// TIA Portal V17 export
// export: Created 2023-02-14T02:49:53.8743835Z, ExportSetting WithDefaults, DisplayName Totally Integrated Automation Portal, DisplayVersion V17, DisplayName TIA Portal Openness, DisplayVersion V17, DisplayName TIA Portal Teamcenter Gateway, DisplayVersion V17, DisplayName TIA Portal Version Control Interface, DisplayVersion V17, DisplayName SINAMICS Startdrive Advanced, DisplayVersion V17, DisplayName SINAMICS Startdrive G130, G150, S120, S150, SINAMICS MV, S210, DisplayVersion V17, DisplayName SINAMICS Startdrive G110M, G120, G120C, G120D, G120P, G115D, DisplayVersion V17, DisplayName STEP 7 Professional, DisplayVersion V17, DisplayName STEP 7 Safety, DisplayVersion V17, DisplayName WinCC Professional, DisplayVersion V17
VAR_GLOBAL   // PLC tag table "RIO Homomixer Panel"
   "FT-12.01 Pulse" AT %I6.0 : Bool;   // PULSE FLOW METER PROCESS WATER
   "FT-12.02 Pulse" AT %I6.1 : Bool;   // PULSE FLOW METER HOT WATER
   "FT-12.01 Flowrate" AT %IW7 : Int;   // FLOW METER PROCESS WATER
   "FT-12.02 Flowrate" AT %IW9 : Int;   // FLOW METER HOT WATER
   "Homo spare 18" AT %IW11 : Int;
   "Homo spare 19" AT %IW13 : Int;
   "ZSC-12.01" AT %I4.0 : Bool;   // INLET PROCESS WATER HOMOMIXER T-12.00 VALVE CLOSE POSITION
   "ZSC-12.02" AT %I4.1 : Bool;   // INLET HOT WATER HOMOMIXER T-12.00 VALVE CLOSE POSITION
   "ZSC-13.01" AT %I4.2 : Bool;   // INLET PROCESS WATER HOMOMIXER T-13.00 VALVE CLOSE POSITION
   "ZSC-13.02" AT %I4.3 : Bool;   // INLET HOT WATER HOMOMIXER T-13.00 VALVE CLOSE POSITION
   "LL-12.01" AT %I4.4 : Bool;   // LOW LEVEL SENSOR HOMOMIXER T-12.00
   "LL-13.01" AT %I4.5 : Bool;   // LOW LEVEL SENSOR HOMOMIXER T-13.00
   "ES1 Homomixer" AT %I4.6 : Bool;   // EMERGENCY STOP RIO HOMOMIXER
   "PS-01 Homomixer" AT %I4.7 : Bool;   // PRESURE SWITCH PNEUMATIC VALVE
   "ZSC-14.01" AT %I5.0 : Bool;   // MAIN CIP SUPPLY HOMOMIXER T-14.00 VALVE CLOSE POSITION
   "ZSC-14.02" AT %I5.1 : Bool;   // MAIN CIP SUPPLY LINE HOMOMIXER T-14.00 VALVE CLOSE POSITION
   "LL-14.01" AT %I5.2 : Bool;   // LOW LEVEL SENSOR HOMOMIXER T-14.00
   "Homo spare 01" AT %I5.3 : Bool;
   "Homo spare 02" AT %I5.4 : Bool;
   "Homo spare 03" AT %I5.5 : Bool;
   "Homo spare 04" AT %I5.6 : Bool;
   "Homo spare 05" AT %I5.7 : Bool;
   "Homo spare 06" AT %I6.2 : Bool;
   "Homo spare 07" AT %I6.3 : Bool;
   "Homo spare 08" AT %I6.4 : Bool;
   "Homo spare 09" AT %I6.5 : Bool;
   "Homo spare 10" AT %I6.6 : Bool;
   "Homo spare 11" AT %I6.7 : Bool;
   "Start/Stop P-12.01" AT %Q2.0 : Bool;   // START/STOP DIAPHRAGM PUMP HOMOMIXER T-12.00
   "Start/Stop P-13.01" AT %Q2.1 : Bool;   // START/STOP DIAPHRAGM PUMP HOMOMIXER T-13.00
   "Start/Stop P-14.01" AT %Q2.2 : Bool;   // START/STOP DIAPHRAGM PUMP HOMOMIXER T-14.00
   "Homo spare 13" AT %Q2.3 : Bool;
   "Homo spare 14" AT %Q2.4 : Bool;
   "Homo spare 15" AT %Q2.5 : Bool;
   "Homo spare 16" AT %Q2.6 : Bool;
   "Homo spare 17" AT %Q2.7 : Bool;
   "AV-12.01" AT %Q22.0 : Bool;   // AUTO BUTTERFLY VALVE PW INLET TO HOMOMIXER T-12.00
   "AV-12.02" AT %Q22.1 : Bool;   // AUTO BUTTERFLY VALVE HOT WATER INLET TO HOMOMIXER T-12.00
   "AV-12.03" AT %Q22.2 : Bool;   // AUTO BUTTERFLY VALVE OUTLET FROM HOMOMIXER T-12.00
   "AV-12.04" AT %Q22.3 : Bool;   // AUTO BUTTERFLY VALVE CIP SUPPLY LINE T-12.00 FROM DP-12.01
   "AV-12.05" AT %Q22.4 : Bool;   // AUTO BUTTERFLY VALVE CIP RETURN FROM HOMOMIXER T-12.00
   "AV-12.06" AT %Q22.5 : Bool;   // AUTO BUTTERFLY VALVE BYPASS DIAPRAGM PUMP P-12.01
   "AV-12.07" AT %Q22.6 : Bool;   // AUTO BUTTERFLY VALVE CIP SUPPLY HOMOMIXER T-12.00
   "AV-12.11" AT %Q22.7 : Bool;   // AUTO BUTTERFLY VALVE MAIN CIP SUPPLY LINE 1 HOMOMIXER T-12.00
   "AV-12.12" AT %Q23.0 : Bool;   // AUTO BUTTERFLY VALVE MAIN CIP SUPPLY LINE 1 HOT WATER T-01.00
   "AV-13.01" AT %Q23.1 : Bool;   // AUTO BUTTERFLY VALVE PW INLET TO HOMOMIXER T-13.00
   "AV-13.02" AT %Q23.2 : Bool;   // AUTO BUTTERFLY VALVE HOT WATER INLET TO HOMOMIXER T-13.00
   "AV-13.03" AT %Q23.3 : Bool;   // AUTO BUTTERFLY VALVE OUTLET FROM HOMOMIXER T-13.00
   "AV-13.04" AT %Q23.4 : Bool;   // AUTO BUTTERFLY VALVE CIP SUPPLY LINE T-13.00 FROM DP-12.01
   "AV-13.05" AT %Q23.5 : Bool;   // AUTO BUTTERFLY VALVE CIP RETURN FROM HOMOMIXER T-13.00
   "AV-13.06" AT %Q23.6 : Bool;   // AUTO BUTTERFLY VALVE BYPASS DIAPRAGM PUMP P-13.01
   "AV-13.07" AT %Q23.7 : Bool;   // AUTO BUTTERFLY VALVE CIP SUPPLY HOMOMIXER T-13.00
   "AV-14.01" AT %Q24.0 : Bool;   // AUTO BUTTERFLY VALVE PW INLET TO HOMOMIXER T-14.00
   "AV-14.02" AT %Q24.1 : Bool;   // AUTO BUTTERFLY VALVE HOT WATER INLET TO HOMOMIXER T-14.00
   "AV-14.03" AT %Q24.2 : Bool;   // AUTO BUTTERFLY VALVE OUTLET FROM HOMOMIXER T-14.00
   "AV-14.04" AT %Q24.3 : Bool;   // AUTO BUTTERFLY VALVE CIP SUPPLY LINE T-14.00 CIP SUPPLY LINE 1
   "AV-14.05" AT %Q24.4 : Bool;   // AUTO BUTTERFLY VALVE CIP RETURN FROM HOMOMIXER T-14.00
   "AV-14.06" AT %Q24.5 : Bool;   // AUTO BUTTERFLY VALVE BYPASS DIAPRAGM PUMP P-14.01
   "AV-14.07" AT %Q24.6 : Bool;   // AUTO BUTTERFLY VALVE CIP SUPPLY HOMOMIXER T-14.00
END_VAR
